// SIMATIC S7-200 project (STEP 7-Micro/WIN), CPU 224XP REL 02.00

ORGANIZATION_BLOCK 主程序:OB1
TITLE=计算最近一小时的累计值
BEGIN
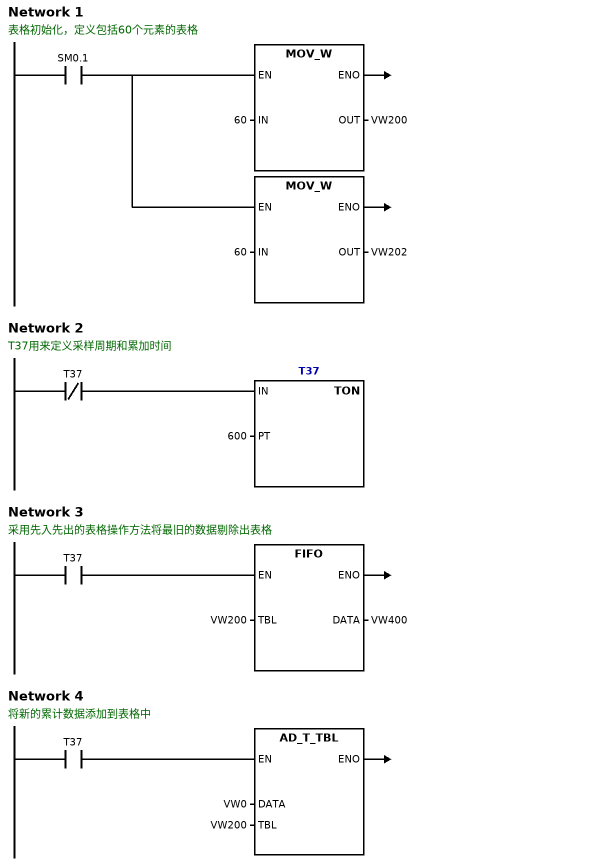
Network 1
// 表格初始化，定义包括60个元素的表格
// (network saved uncompiled; LAD cells follow)
// row 0: c0 -| |- SM0.1 v  c1 --  c2 [MOV_W EN:=power@row0, IN:=60, ENO=>power, OUT=>VW200]  c3 ->
// row 1: c0 ^v  c2 [box]
// row 2: c0 ^  c1 --  c2 [MOV_W EN:=power@row2, IN:=60, ENO=>power, OUT=>VW202]  c3 ->
// row 3: c2 [box]
Network 2
// T37用来定义采样周期和累加时间
// (network saved uncompiled; LAD cells follow)
// row 0: c0 -|/|- T37  c1 --  c2 [TON T37 IN:=power@row0, PT:=600]
// row 1: c2 [box]
Network 3
// 采用先入先出的表格操作方法将最旧的数据剔除出表格
LD     T37
FIFO   VW200, VW400
Network 4
// 将新的累计数据添加到表格中
LD     T37
ATT    VW0, VW200
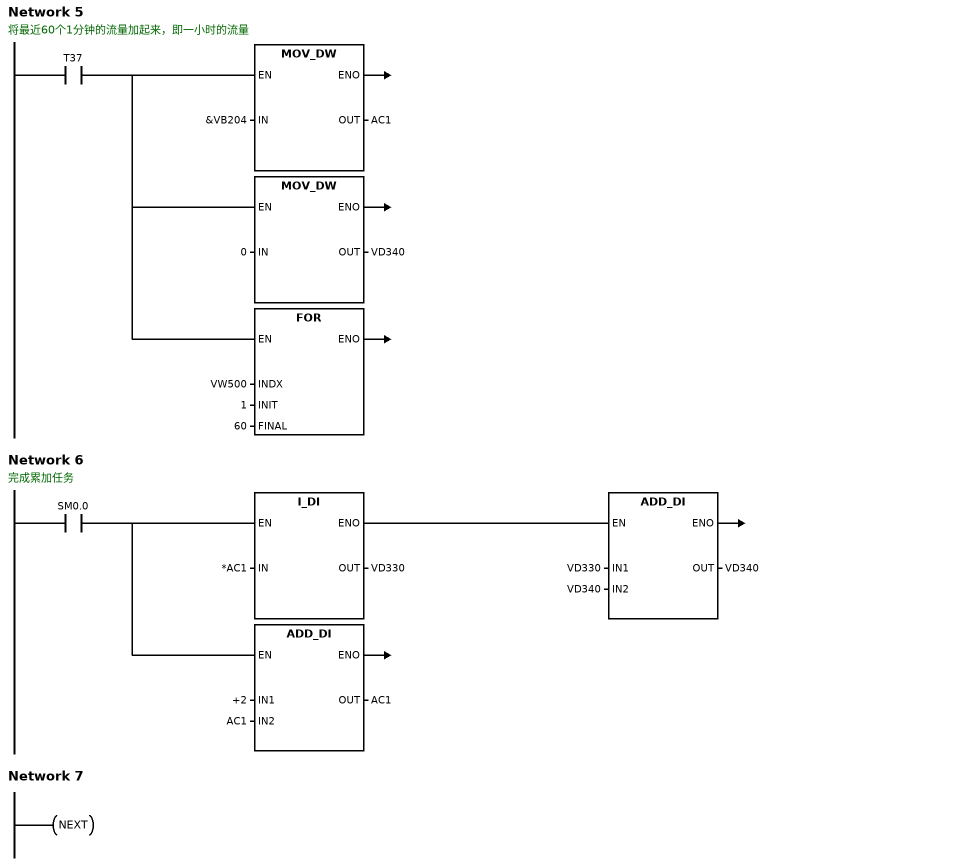
Network 5
// 将最近60个1分钟的流量加起来，即一小时的流量
// (network saved uncompiled; LAD cells follow)
// row 0: c0 -| |- T37 v  c1 --  c2 [MOV_DW EN:=power@row0, IN:=&VB204, ENO=>power, OUT=>AC1]  c3 ->
// row 1: c0 ^v  c2 [box]
// row 2: c0 ^v  c1 --  c2 [MOV_DW EN:=power@row2, IN:=0, ENO=>power, OUT=>VD340]  c3 ->
// row 3: c0 ^v  c2 [box]
// row 4: c0 ^  c1 --  c2 [FOR EN:=power@row4, INDX:=VW500, INIT:=1, FINAL:=60, ENO=>power]  c3 ->
// row 5: c2 [box]
Network 6
// 完成累加任务
LD     SM0.0
LPS
ITD    *AC1, VD330
AENO
+D     VD330, VD340
LPP
+D     +2, AC1
Network 7
NEXT
END_ORGANIZATION_BLOCK
